{attribute 'qualified_only'}
{attribute 'strict'}
{attribute 'to_string'}
TYPE E_ErrorLevel :
(
	NONE := 0,
	Low,
	High,
	Critical
)UINT;
END_TYPE

(* stored: Version 1.1.0.1, ProductVersion 3.1.4026.18
   DUT E_ErrorLevel: Id {3dafef54-bbd9-4727-8d37-ca137afbc442} *)
